// TIA Portal V17 export
// export: Created 2025-03-07T09:19:49.1205601Z, ExportSetting WithDefaults, DisplayName Totally Integrated Automation Portal, DisplayVersion V17 Update 8, DisplayName TIA Portal Openness, DisplayVersion V17 Update 8, DisplayName TIA Portal Version Control Interface, DisplayVersion V17, DisplayName SINAMICS Startdrive Advanced, DisplayVersion V17 SP2, DisplayName SINAMICS Startdrive G110M, G120, G120C, G120D, G120P, G115D, DisplayVersion V17 SP2, DisplayName SINAMICS Startdrive G130, G150, S120, S150, SINAMICS MV, S210, DisplayVersion V17 SP2, DisplayName STEP 7 Professional, DisplayVersion V17 Update 8, DisplayName SINUMERIK ONE STEP 7 Toolbox, DisplayVersion V17 Update 12, DisplayName SINUMERIK 840D sl STEP 7 Toolbox, DisplayVersion V17 Update 12, DisplayName STEP 7 Safety, DisplayVersion V17 Update 6, DisplayName WinCC Advanced, DisplayVersion V17 Update 8
TYPE "IOL_CONF"
// stored: IsFailsafeCompliant false
   STRUCT
      SELECTED : Struct
         SCRN_1 : Bool;   // SCREEN ONE SELECTED / SCREEN 1 SELECTED
         SCRN_2 : Bool;   // SCREEN TWO SELECTED / SCREEN 2 SELECTED
         SCRN_3 : Bool;   // SCREEN THREE SELECTED / SCREEN 3 SELECTED
         SCRN_4 : Bool;   // SCREEN FOUR SELECTED / SCREEN 4 SELECTED
         SCRN_5 : Bool;   // SCREEN FIVE SELECTED / SCREEN 5 SELECTED
         SCRN_6 : Bool;   // SCREEN SIX SELECTED / SCREEN 6 SELECTED
         SCRN_7 : Bool;   // SCREEN SEVEN SELECTED / SCREEN 7 SELECTED
         SCRN_8 : Bool;   // SCREEN EIGHT SELECTED / SCREEN 8 SELECTED
         SCRN_11 : Bool;   // SCREEN 11 SELECTED
         SCRN_12 : Bool;   // SCREEN 12 SELECTED
         SCRN_13 : Bool;   // SCREEN 13 SELECTED
         SCRN_14 : Bool;   // SCREEN 14 SELECTED
         SCRN_15 : Bool;   // SCREEN 15 SELECTED
         SCRN_16 : Bool;   // SCREEN 16 SELECTED
         SCRN_17 : Bool;   // SCREEN 17 SELECTED
         SCRN_18 : Bool;   // SCREEN 18 SELECTED
      END_STRUCT;
      HMI_VARIABLES : Struct
         DONE : Bool;   // HMI DONE BIT
         BUSY : Bool;   // HMI BUSY BIT
         ERROR : Bool;   // HMI ERROR BIT
         RD_WRT_HMI : Bool;   // HMI BUTTON READ/ WRITE SELECTION
         EXECUTE_ACTION : Bool;   // HMI EXECUTE READ/WRITE
         SPARE_205 : Bool;   // SPARE BIT
         SPARE_206 : Bool;   // SPARE BIT
         SPARE_207 : Bool;   // SPARE BIT
         SPARE_210 : Bool;   // SPARE BIT
         SPARE_211 : Bool;   // SPARE BIT
         SPARE_212 : Bool;   // SPARE BIT
         SPARE_213 : Bool;   // SPARE BIT
         SPARE_214 : Bool;   // SPARE BIT
         SPARE_215 : Bool;   // SPARE BIT
         SPARE_216 : Bool;   // SPARE BIT
         SPARE_217 : Bool;   // SPARE BIT
         IOL_LIST : Int;   // SELECTION LIST
         IO_LIST_OLD : Int;   // SELECTION LIST OLD
         SCRN_NMBR : Int;   // SELECTED SCREEN
         SCRN_NMBR_OLD : Int;   // SELECTED SCREEN OLD
         RND_INTRVL_1 : Real;   // ROUND INTERVAL FIRST VALUE
         RND_INTRVL_2 : Real;   // ROUND INTVERAL SECOND VALUE
         VAR_ERROR : Byte;   // VARIABLE NUMBER ERROR TAKE PLACE
         TOT_FLT : Byte;   // TOTAL FAULT
         FIRST_VALUE_DISPLAY : Real;   // HMI FIRST VALUE DISPLAY
         SECOND_VALUE_DISPLAY : Real;   // HMI SECOND VALUE DISPLAY
         SPARE_DISPLAY0 : Real;   // HMI SPARE DISPLAY
         SPARE_DISPLAY1 : Real;   // HMI SPARE DISPLAY
         SPARE_DISPLAY2 : Real;   // HMI SPARE DISPLAY
         REAL_VALUE : Array[0..17] of Real;   // REAL VALUE
      END_STRUCT;
      SPARE : Array[1..24] of Byte;
      GEOADR { ExternalAccessible := 'False'; ExternalVisible := 'False'; ExternalWritable := 'False'; S7_SetPoint := 'True'} : GEOADDR;   // INFO TO DETERMINE HW_IO
      CONFIG_DATA : Struct
         SPARE : UInt;   // DATA ADDRESS ID / Spare
         DATA_PORT : UInt;   // DATA PORT
         CAP_NMBR : UInt;   // CAP NUMBER
         VAR_RO : UInt;   // READ ONLY VARIABLES
         TOT_REAL_VAR : UInt;   // TOTAL REAL VARIABLES TO READ
         REAL_VAR_ARRAY_POS : UInt;   // REAL VARIABLES FIRST POSITION AT ARRAY
         TOT_VAR_TO_RD : UInt;   // TOTAL VARIABLES TO READ
      END_STRUCT;
      IOL_CONF : Array[1..20] of Struct
         INDX : Int;   // INDEX
         SBINDX : Int;   // SUBINDEX
         LNG : Int;   // LENGTH
         GRDNT : Real;   // GRADIENT
         OFFST : Real;   // OFFSET
         ROUND_1_OR_2 : Int;   // ROUND INTERVAL TO USE 1 OR 2
      END_STRUCT;
   END_STRUCT;
   // // GEOADR.HWTYPE : HW type (info to obtain from hw component) 4=module
   // // GEOADR.AREA : Normally not used
   // // GEOADR.IOSYSTEM : Network the IO master is on (100 profinet)(Normally always 100)
   // // GEOADR.STATION : Device No. of the IO master in hardware
   // // GEOADR.SLOT : Slot Number in hardware
   // // GEOADR.SUBSLOT : Sub Slot Number if necessary (Normally not used)
END_TYPE
